TYPE TcoKrc4_IO_v_5_x_x :
STRUCT
	PnIoBoxState AT %I*	:	UINT;
	PnIoBoxDiag AT %I*	:	UINT;
	PnIoBoxCtrl AT %Q*	:	UINT;
	{attribute addProperty Name "<#IN#>"}
	In : TcoKrc4_Inputs_v_5_x_x;
	{attribute addProperty Name "<#OUT#>"}
	Out : TcoKrc4_Outputs_v_5_x_x;
END_STRUCT
END_TYPE

(* stored: Version 1.1.0.1, ProductVersion 3.1.4024.12
   DUT TcoKrc4_IO_v_5_x_x: Id {a959940f-68ff-0922-2b75-acf3bc5a30c8} *)
